VAR_GLOBAL PERSISTENT
	
/////////////////////////////////////////////////////////////////////////////////////Log/////////////////////////////////////////////////////////////////////////////////////
	
	stUserLog					: ARRAY [0..250] OF ST_UserLog;
	
	stStatisticsHMI				: ARRAY [0..3] OF ST_StatisticsHMI;	//0: GENERAL
																	//1: STATION 1
																	//2: STATION 2
																	//3: STATION 3
	aDataHistory				: ARRAY[0..200] OF ST_CycleData;
	nIndexDataHistory			: DINT;
	astEventsHistory			: ARRAY[0..200] OF ST_EventsHistory;


END_VAR

(* stored: Version 1.1.0.1, ProductVersion 3.1.4024.13
   GVL GVL_Persistent: Id {c4d03ea6-35af-4633-972d-fef3cfe7daa9} *)
